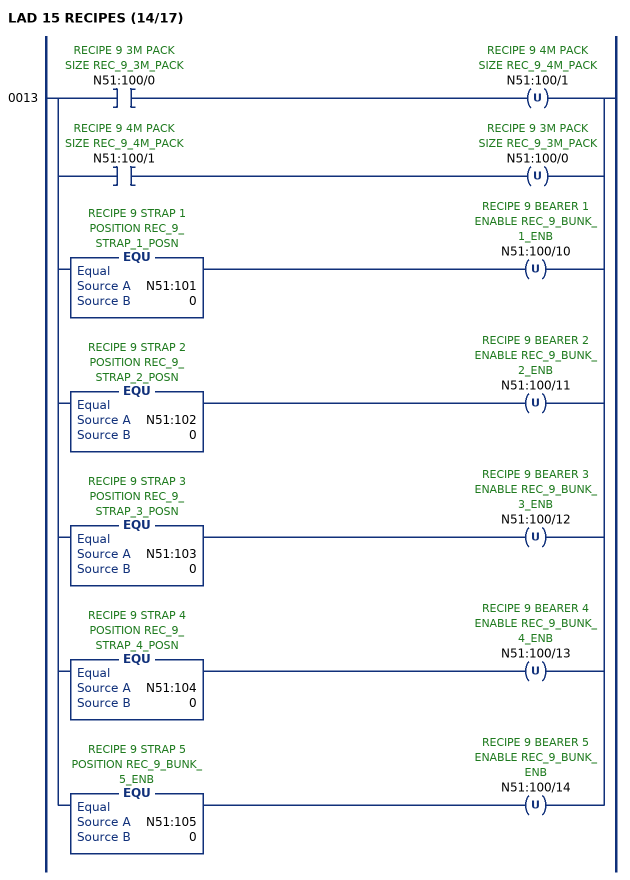
% Rung: 13 %
SOR BST XIC N51:100/0 OTU N51:100/1 NXB XIC N51:100/1 OTU N51:100/0 NXB EQU N51:101 0 OTU N51:100/10 NXB EQU N51:102 0 OTU N51:100/11 NXB EQU N51:103 0 OTU N51:100/12 NXB EQU N51:104 0 OTU N51:100/13 NXB EQU N51:105 0 OTU N51:100/14 BND EOR
%   N51:100/0  REC_9_3M_PACK  "RECIPE 9 3M PACK SIZE" %
%   N51:100/1  REC_9_4M_PACK  "RECIPE 9 4M PACK SIZE" %
%   N51:101  REC_9_STRAP_1_POSN  "RECIPE 9 STRAP 1 POSITION" %
%   N51:100/10  REC_9_BUNK_1_ENB  "RECIPE 9 BEARER 1 ENABLE" %
%   N51:102  REC_9_STRAP_2_POSN  "RECIPE 9 STRAP 2 POSITION" %
%   N51:100/11  REC_9_BUNK_2_ENB  "RECIPE 9 BEARER 2 ENABLE" %
%   N51:103  REC_9_STRAP_3_POSN  "RECIPE 9 STRAP 3 POSITION" %
%   N51:100/12  REC_9_BUNK_3_ENB  "RECIPE 9 BEARER 3 ENABLE" %
%   N51:104  REC_9_STRAP_4_POSN  "RECIPE 9 STRAP 4 POSITION" %
%   N51:100/13  REC_9_BUNK_4_ENB  "RECIPE 9 BEARER 4 ENABLE" %
%   N51:105  REC_9_BUNK_5_ENB  "RECIPE 9 STRAP 5 POSITION" %
%   N51:100/14  REC_9_BUNK_ENB  "RECIPE 9 BEARER 5 ENABLE" %

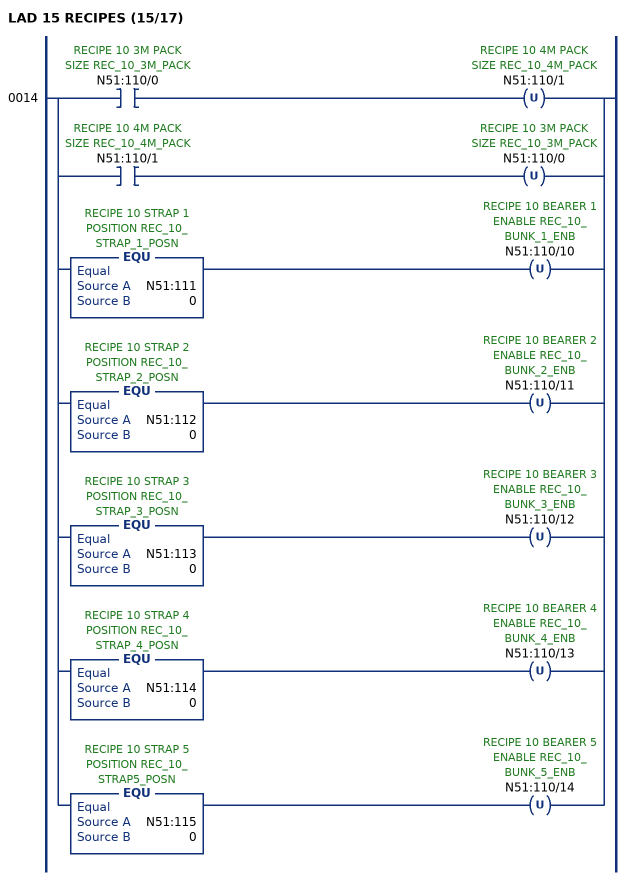
% Rung: 14 %
SOR BST XIC N51:110/0 OTU N51:110/1 NXB XIC N51:110/1 OTU N51:110/0 NXB EQU N51:111 0 OTU N51:110/10 NXB EQU N51:112 0 OTU N51:110/11 NXB EQU N51:113 0 OTU N51:110/12 NXB EQU N51:114 0 OTU N51:110/13 NXB EQU N51:115 0 OTU N51:110/14 BND EOR
%   N51:110/0  REC_10_3M_PACK  "RECIPE 10 3M PACK SIZE" %
%   N51:110/1  REC_10_4M_PACK  "RECIPE 10 4M PACK SIZE" %
%   N51:111  REC_10_STRAP_1_POSN  "RECIPE 10 STRAP 1 POSITION" %
%   N51:110/10  REC_10_BUNK_1_ENB  "RECIPE 10 BEARER 1 ENABLE" %
%   N51:112  REC_10_STRAP_2_POSN  "RECIPE 10 STRAP 2 POSITION" %
%   N51:110/11  REC_10_BUNK_2_ENB  "RECIPE 10 BEARER 2 ENABLE" %
%   N51:113  REC_10_STRAP_3_POSN  "RECIPE 10 STRAP 3 POSITION" %
%   N51:110/12  REC_10_BUNK_3_ENB  "RECIPE 10 BEARER 3 ENABLE" %
%   N51:114  REC_10_STRAP_4_POSN  "RECIPE 10 STRAP 4 POSITION" %
%   N51:110/13  REC_10_BUNK_4_ENB  "RECIPE 10 BEARER 4 ENABLE" %
%   N51:115  REC_10_STRAP5_POSN  "RECIPE 10 STRAP 5 POSITION" %
%   N51:110/14  REC_10_BUNK_5_ENB  "RECIPE 10 BEARER 5 ENABLE" %

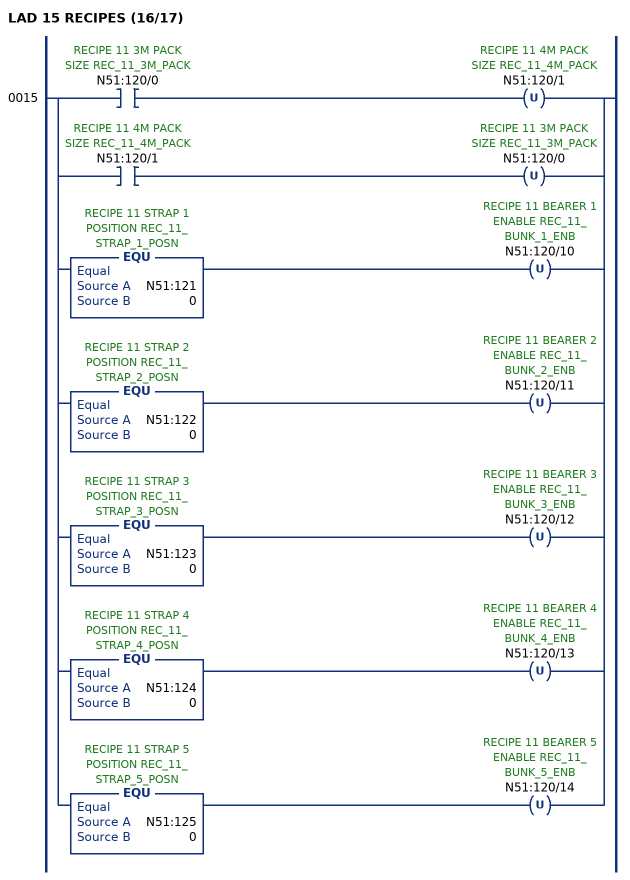
% Rung: 15 %
SOR BST XIC N51:120/0 OTU N51:120/1 NXB XIC N51:120/1 OTU N51:120/0 NXB EQU N51:121 0 OTU N51:120/10 NXB EQU N51:122 0 OTU N51:120/11 NXB EQU N51:123 0 OTU N51:120/12 NXB EQU N51:124 0 OTU N51:120/13 NXB EQU N51:125 0 OTU N51:120/14 BND EOR
%   N51:120/0  REC_11_3M_PACK  "RECIPE 11 3M PACK SIZE" %
%   N51:120/1  REC_11_4M_PACK  "RECIPE 11 4M PACK SIZE" %
%   N51:121  REC_11_STRAP_1_POSN  "RECIPE 11 STRAP 1 POSITION" %
%   N51:120/10  REC_11_BUNK_1_ENB  "RECIPE 11 BEARER 1 ENABLE" %
%   N51:122  REC_11_STRAP_2_POSN  "RECIPE 11 STRAP 2 POSITION" %
%   N51:120/11  REC_11_BUNK_2_ENB  "RECIPE 11 BEARER 2 ENABLE" %
%   N51:123  REC_11_STRAP_3_POSN  "RECIPE 11 STRAP 3 POSITION" %
%   N51:120/12  REC_11_BUNK_3_ENB  "RECIPE 11 BEARER 3 ENABLE" %
%   N51:124  REC_11_STRAP_4_POSN  "RECIPE 11 STRAP 4 POSITION" %
%   N51:120/13  REC_11_BUNK_4_ENB  "RECIPE 11 BEARER 4 ENABLE" %
%   N51:125  REC_11_STRAP_5_POSN  "RECIPE 11 STRAP 5 POSITION" %
%   N51:120/14  REC_11_BUNK_5_ENB  "RECIPE 11 BEARER 5 ENABLE" %

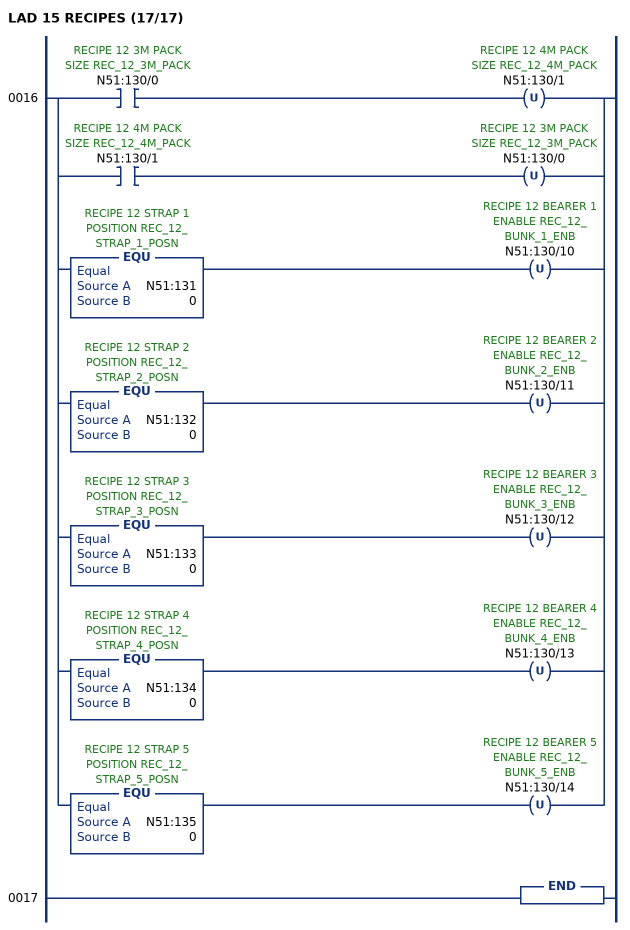
% Rung: 16 %
SOR BST XIC N51:130/0 OTU N51:130/1 NXB XIC N51:130/1 OTU N51:130/0 NXB EQU N51:131 0 OTU N51:130/10 NXB EQU N51:132 0 OTU N51:130/11 NXB EQU N51:133 0 OTU N51:130/12 NXB EQU N51:134 0 OTU N51:130/13 NXB EQU N51:135 0 OTU N51:130/14 BND EOR
%   N51:130/0  REC_12_3M_PACK  "RECIPE 12 3M PACK SIZE" %
%   N51:130/1  REC_12_4M_PACK  "RECIPE 12 4M PACK SIZE" %
%   N51:131  REC_12_STRAP_1_POSN  "RECIPE 12 STRAP 1 POSITION" %
%   N51:130/10  REC_12_BUNK_1_ENB  "RECIPE 12 BEARER 1 ENABLE" %
%   N51:132  REC_12_STRAP_2_POSN  "RECIPE 12 STRAP 2 POSITION" %
%   N51:130/11  REC_12_BUNK_2_ENB  "RECIPE 12 BEARER 2 ENABLE" %
%   N51:133  REC_12_STRAP_3_POSN  "RECIPE 12 STRAP 3 POSITION" %
%   N51:130/12  REC_12_BUNK_3_ENB  "RECIPE 12 BEARER 3 ENABLE" %
%   N51:134  REC_12_STRAP_4_POSN  "RECIPE 12 STRAP 4 POSITION" %
%   N51:130/13  REC_12_BUNK_4_ENB  "RECIPE 12 BEARER 4 ENABLE" %
%   N51:135  REC_12_STRAP_5_POSN  "RECIPE 12 STRAP 5 POSITION" %
%   N51:130/14  REC_12_BUNK_5_ENB  "RECIPE 12 BEARER 5 ENABLE" %
% Rung: 17 %
SOR END EOR

LADDER 16 "ENCODER"    % ENCODER %
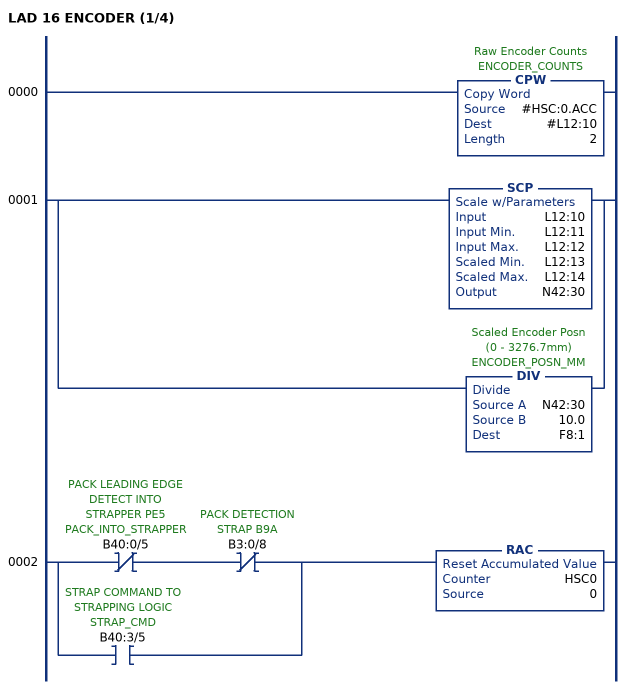
% Rung: 0 %
SOR CPW #HSC:0.ACC #L12:10 2 EOR
%   L12:10  ENCODER_COUNTS  "Raw Encoder Counts" %
% Rung: 1 %
SOR BST SCP L12:10 L12:11 L12:12 L12:13 L12:14 N42:30 NXB DIV N42:30 10.0 F8:1 BND EOR
%   L12:10  ENCODER_COUNTS  "Raw Encoder Counts" %
%   F8:1  ENCODER_POSN_MM  "Scaled Encoder Posn (0 - 3276.7mm)" %
% Rung: 2 %
SOR BST XIO B40:0/5 XIO B3:0/8 NXB XIC B40:3/5 BND RAC HSC0 0 EOR
%   B40:0/5  PACK_INTO_STRAPPER  "PACK LEADING EDGE DETECT INTO STRAPPER PE5" %
%   B3:0/8  B9A  "PACK DETECTION STRAP" %
%   B40:3/5  STRAP_CMD  "STRAP COMMAND TO STRAPPING LOGIC" %

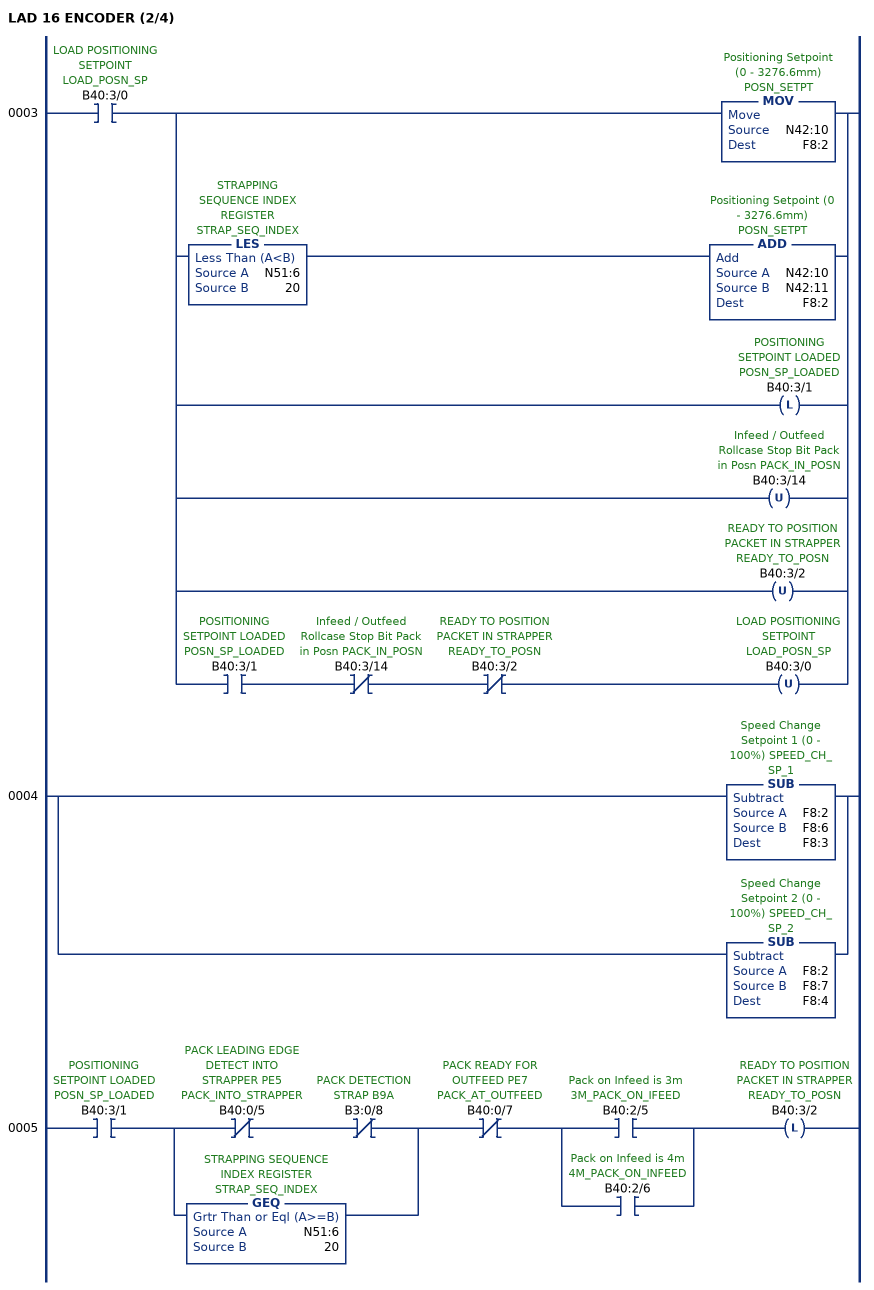
% Rung: 3 %
SOR XIC B40:3/0 BST MOV N42:10 F8:2 NXB LES N51:6 20 ADD N42:10 N42:11 F8:2 NXB OTL B40:3/1 NXB OTU B40:3/14 NXB OTU B40:3/2 NXB XIC B40:3/1 XIO B40:3/14 XIO B40:3/2 OTU B40:3/0 BND EOR
%   B40:3/0  LOAD_POSN_SP  "LOAD POSITIONING SETPOINT" %
%   N42:10  POSN_SETPOINT  "POSITIONING SETPOINT" %
%   F8:2  POSN_SETPT  "Positioning Setpoint (0 - 3276.6mm)" %
%   N51:6  STRAP_SEQ_INDEX  "STRAPPING SEQUENCE INDEX REGISTER" %
%   N42:11  POSN_SP_OFFSET  "Positioning Setpoint Offset" %
%   B40:3/1  POSN_SP_LOADED  "POSITIONING SETPOINT LOADED" %
%   B40:3/14  PACK_IN_POSN  "Infeed / Outfeed Rollcase Stop Bit Pack in Posn" %
%   B40:3/2  READY_TO_POSN  "READY TO POSITION PACKET IN STRAPPER" %
% Rung: 4 %
SOR BST SUB F8:2 F8:6 F8:3 NXB SUB F8:2 F8:7 F8:4 BND EOR
%   F8:2  POSN_SETPT  "Positioning Setpoint (0 - 3276.6mm)" %
%   F8:6  SP_CHANGE_FACT_1  "Speed Change Position Factor 1" %
%   F8:3  SPEED_CH_SP_1  "Speed Change Setpoint 1 (0 - 100%)" %
%   F8:7  SP_CHANGE_FACT_2  "Speed Change Positon Factor 2" %
%   F8:4  SPEED_CH_SP_2  "Speed Change Setpoint 2 (0 - 100%)" %
% Rung: 5 %
SOR XIC B40:3/1 BST XIO B40:0/5 XIO B3:0/8 NXB GEQ N51:6 20 BND XIO B40:0/7 BST XIC B40:2/5 NXB XIC B40:2/6 BND OTL B40:3/2 EOR
%   B40:3/1  POSN_SP_LOADED  "POSITIONING SETPOINT LOADED" %
%   B40:0/5  PACK_INTO_STRAPPER  "PACK LEADING EDGE DETECT INTO STRAPPER PE5" %
%   B3:0/8  B9A  "PACK DETECTION STRAP" %
%   N51:6  STRAP_SEQ_INDEX  "STRAPPING SEQUENCE INDEX REGISTER" %
%   B40:0/7  PACK_AT_OUTFEED  "PACK READY FOR OUTFEED PE7" %
%   B40:2/5  3M_PACK_ON_IFEED  "Pack on Infeed is 3m" %
%   B40:2/6  4M_PACK_ON_INFEED  "Pack on Infeed is 4m" %
%   B40:3/2  READY_TO_POSN  "READY TO POSITION PACKET IN STRAPPER" %

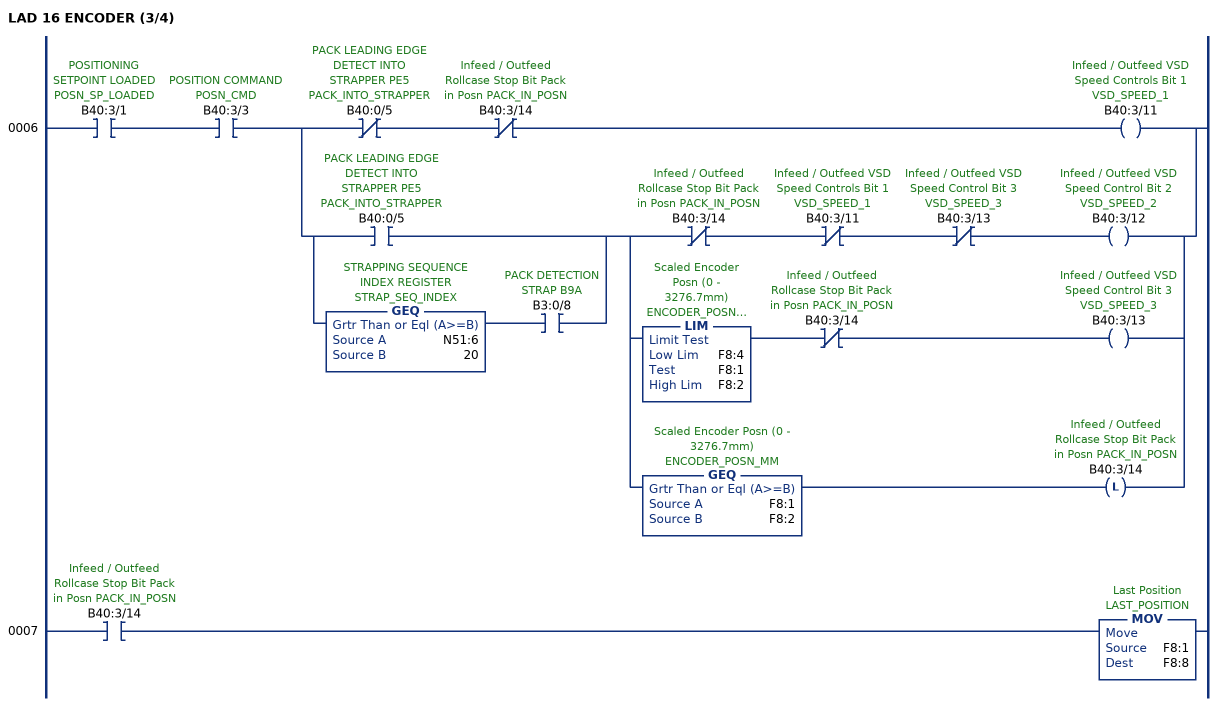
% Rung: 6 %
SOR XIC B40:3/1 XIC B40:3/3 BST XIO B40:0/5 XIO B40:3/14 OTE B40:3/11 NXB BST XIC B40:0/5 NXB GEQ N51:6 20 XIC B3:0/8 BND BST XIO B40:3/14 XIO B40:3/11 XIO B40:3/13 OTE B40:3/12 NXB LIM F8:4 F8:1 F8:2 XIO B40:3/14 OTE B40:3/13 NXB GEQ F8:1 F8:2 OTL B40:3/14 BND BND EOR
%   B40:3/1  POSN_SP_LOADED  "POSITIONING SETPOINT LOADED" %
%   B40:3/3  POSN_CMD  "POSITION COMMAND" %
%   B40:0/5  PACK_INTO_STRAPPER  "PACK LEADING EDGE DETECT INTO STRAPPER PE5" %
%   B40:3/14  PACK_IN_POSN  "Infeed / Outfeed Rollcase Stop Bit Pack in Posn" %
%   B40:3/11  VSD_SPEED_1  "Infeed / Outfeed VSD Speed Controls Bit 1" %
%   N51:6  STRAP_SEQ_INDEX  "STRAPPING SEQUENCE INDEX REGISTER" %
%   B3:0/8  B9A  "PACK DETECTION STRAP" %
%   B40:3/13  VSD_SPEED_3  "Infeed / Outfeed VSD Speed Control Bit 3" %
%   B40:3/12  VSD_SPEED_2  "Infeed / Outfeed VSD Speed Control Bit 2" %
%   F8:4  SPEED_CH_SP_2  "Speed Change Setpoint 2 (0 - 100%)" %
%   F8:1  ENCODER_POSN_MM  "Scaled Encoder Posn (0 - 3276.7mm)" %
%   F8:2  POSN_SETPT  "Positioning Setpoint (0 - 3276.6mm)" %
% Rung: 7 %
SOR XIC B40:3/14 MOV F8:1 F8:8 EOR
%   B40:3/14  PACK_IN_POSN  "Infeed / Outfeed Rollcase Stop Bit Pack in Posn" %
%   F8:1  ENCODER_POSN_MM  "Scaled Encoder Posn (0 - 3276.7mm)" %
%   F8:8  LAST_POSITION  "Last Position" %

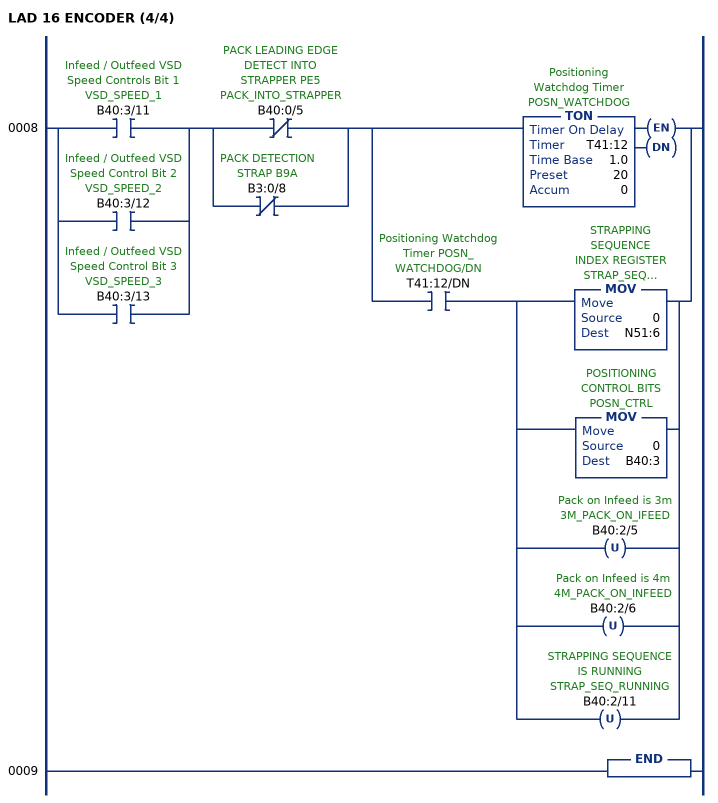
% Rung: 8 %
SOR BST XIC B40:3/11 NXB XIC B40:3/12 NXB XIC B40:3/13 BND BST XIO B40:0/5 NXB XIO B3:0/8 BND BST TON T41:12 1.0 20 0 NXB XIC T41:12/DN BST MOV 0 N51:6 NXB MOV 0 B40:3 NXB OTU B40:2/5 NXB OTU B40:2/6 NXB OTU B40:2/11 BND BND EOR
%   B40:3/11  VSD_SPEED_1  "Infeed / Outfeed VSD Speed Controls Bit 1" %
%   B40:3/12  VSD_SPEED_2  "Infeed / Outfeed VSD Speed Control Bit 2" %
%   B40:3/13  VSD_SPEED_3  "Infeed / Outfeed VSD Speed Control Bit 3" %
%   B40:0/5  PACK_INTO_STRAPPER  "PACK LEADING EDGE DETECT INTO STRAPPER PE5" %
%   B3:0/8  B9A  "PACK DETECTION STRAP" %
%   T41:12  POSN_WATCHDOG  "Positioning Watchdog Timer" %
%   N51:6  STRAP_SEQ_INDEX  "STRAPPING SEQUENCE INDEX REGISTER" %
%   B40:3  POSN_CTRL  "POSITIONING CONTROL BITS" %
%   B40:2/5  3M_PACK_ON_IFEED  "Pack on Infeed is 3m" %
%   B40:2/6  4M_PACK_ON_INFEED  "Pack on Infeed is 4m" %
%   B40:2/11  STRAP_SEQ_RUNNING  "STRAPPING SEQUENCE IS RUNNING" %
% Rung: 9 %
SOR END EOR

LADDER 17 "VSD"    % INFEED VSD'S %
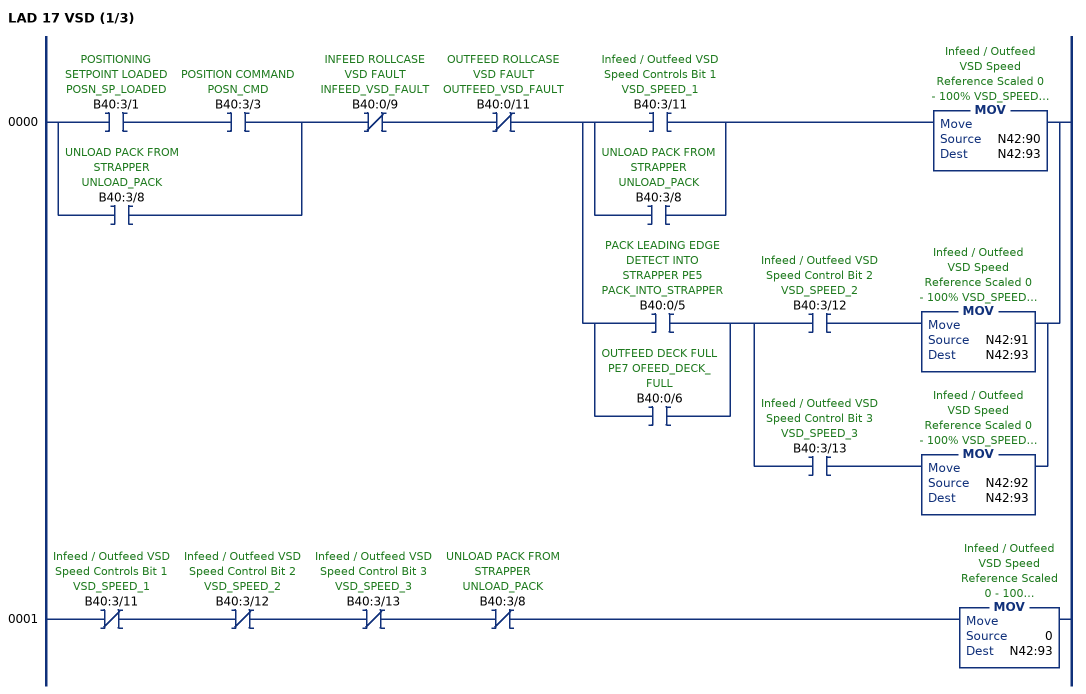
% Rung: 0 %
SOR BST XIC B40:3/1 XIC B40:3/3 NXB XIC B40:3/8 BND XIO B40:0/9 XIO B40:0/11 BST BST XIC B40:3/11 NXB XIC B40:3/8 BND MOV N42:90 N42:93 NXB BST XIC B40:0/5 NXB XIC B40:0/6 BND BST XIC B40:3/12 MOV N42:91 N42:93 NXB XIC B40:3/13 MOV N42:92 N42:93 BND BND EOR
%   B40:3/1  POSN_SP_LOADED  "POSITIONING SETPOINT LOADED" %
%   B40:3/3  POSN_CMD  "POSITION COMMAND" %
%   B40:3/8  UNLOAD_PACK  "UNLOAD PACK FROM STRAPPER" %
%   B40:0/9  INFEED_VSD_FAULT  "INFEED ROLLCASE VSD FAULT" %
%   B40:0/11  OUTFEED_VSD_FAULT  "OUTFEED ROLLCASE VSD FAULT" %
%   B40:3/11  VSD_SPEED_1  "Infeed / Outfeed VSD Speed Controls Bit 1" %
%   N42:90  VSD_SPEED_SP_1  "Infeed / Outfeed VSD Speed Setpoint 1 (0 - 100%)" %
%   N42:93  VSD_SPEED_REF  "Infeed / Outfeed VSD Speed Reference Scaled 0 - 100%" %
%   B40:0/5  PACK_INTO_STRAPPER  "PACK LEADING EDGE DETECT INTO STRAPPER PE5" %
%   B40:0/6  OFEED_DECK_FULL  "OUTFEED DECK FULL PE7" %
%   B40:3/12  VSD_SPEED_2  "Infeed / Outfeed VSD Speed Control Bit 2" %
%   N42:91  VSD_SPEED_SP_2  "Infeed / Outfeed VSD Speed Setpoint 2 (0 - 100%)" %
%   B40:3/13  VSD_SPEED_3  "Infeed / Outfeed VSD Speed Control Bit 3" %
%   N42:92  VSD_SPEED_SP_3  "Infeed / Outfeed VSD Speed Setpoint 3 (0 - 100%)" %
% Rung: 1 %
SOR XIO B40:3/11 XIO B40:3/12 XIO B40:3/13 XIO B40:3/8 MOV 0 N42:93 EOR
%   B40:3/11  VSD_SPEED_1  "Infeed / Outfeed VSD Speed Controls Bit 1" %
%   B40:3/12  VSD_SPEED_2  "Infeed / Outfeed VSD Speed Control Bit 2" %
%   B40:3/13  VSD_SPEED_3  "Infeed / Outfeed VSD Speed Control Bit 3" %
%   B40:3/8  UNLOAD_PACK  "UNLOAD PACK FROM STRAPPER" %
%   N42:93  VSD_SPEED_REF  "Infeed / Outfeed VSD Speed Reference Scaled 0 - 100%" %

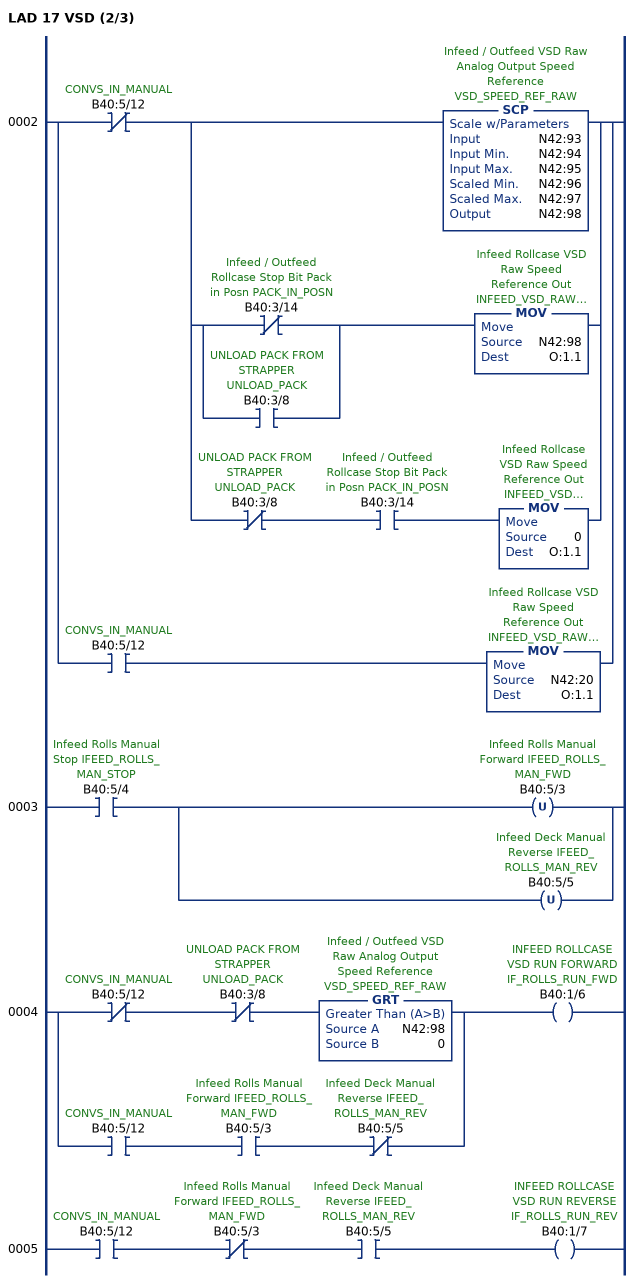
% Rung: 2 %
SOR BST XIO B40:5/12 BST BST SCP N42:93 N42:94 N42:95 N42:96 N42:97 N42:98 NXB BST XIO B40:3/14 NXB XIC B40:3/8 BND MOV N42:98 O:1.1 BND NXB XIO B40:3/8 XIC B40:3/14 MOV 0 O:1.1 BND NXB XIC B40:5/12 MOV N42:20 O:1.1 BND EOR
%   B40:5/12  CONVS_IN_MANUAL %
%   N42:93  VSD_SPEED_REF  "Infeed / Outfeed VSD Speed Reference Scaled 0 - 100%" %
%   N42:94  "Infeed / Outfeed VSD Scaled Input Max" %
%   N42:95  "Infeed / Outfeed VSD Scaled Input Min" %
%   N42:96  "Infeed / Outfeed VSD Scaled Output Min To Analog" %
%   N42:97  "Infeed / Outfeed VSD Scaled Output Max To Analog" %
%   N42:98  VSD_SPEED_REF_RAW  "Infeed / Outfeed VSD Raw Analog Output Speed Reference" %
%   B40:3/14  PACK_IN_POSN  "Infeed / Outfeed Rollcase Stop Bit Pack in Posn" %
%   B40:3/8  UNLOAD_PACK  "UNLOAD PACK FROM STRAPPER" %
%   O:1.1  INFEED_VSD_RAW_OUT  "Infeed Rollcase VSD Raw Speed Reference Out" %
%   N42:20  VSD_MAN_SPEED_SP  "VSD MANUAL SPEED SETPOINT" %
% Rung: 3 %
SOR XIC B40:5/4 BST OTU B40:5/3 NXB OTU B40:5/5 BND EOR
%   B40:5/4  IFEED_ROLLS_MAN_STOP  "Infeed Rolls Manual Stop" %
%   B40:5/3  IFEED_ROLLS_MAN_FWD  "Infeed Rolls Manual Forward" %
%   B40:5/5  IFEED_ROLLS_MAN_REV  "Infeed Deck Manual Reverse" %
% Rung: 4 %
SOR BST XIO B40:5/12 XIO B40:3/8 GRT N42:98 0 NXB XIC B40:5/12 XIC B40:5/3 XIO B40:5/5 BND OTE B40:1/6 EOR
%   B40:5/12  CONVS_IN_MANUAL %
%   B40:3/8  UNLOAD_PACK  "UNLOAD PACK FROM STRAPPER" %
%   N42:98  VSD_SPEED_REF_RAW  "Infeed / Outfeed VSD Raw Analog Output Speed Reference" %
%   B40:5/3  IFEED_ROLLS_MAN_FWD  "Infeed Rolls Manual Forward" %
%   B40:5/5  IFEED_ROLLS_MAN_REV  "Infeed Deck Manual Reverse" %
%   B40:1/6  IF_ROLLS_RUN_FWD  "INFEED ROLLCASE VSD RUN FORWARD" %
% Rung: 5 %
SOR XIC B40:5/12 XIO B40:5/3 XIC B40:5/5 OTE B40:1/7 EOR
%   B40:5/12  CONVS_IN_MANUAL %
%   B40:5/3  IFEED_ROLLS_MAN_FWD  "Infeed Rolls Manual Forward" %
%   B40:5/5  IFEED_ROLLS_MAN_REV  "Infeed Deck Manual Reverse" %
%   B40:1/7  IF_ROLLS_RUN_REV  "INFEED ROLLCASE VSD RUN REVERSE" %

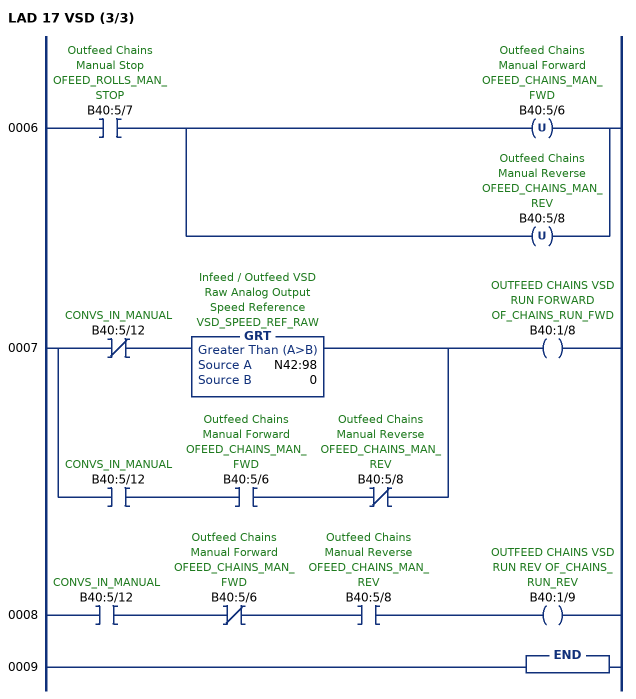
% Rung: 6 %
SOR XIC B40:5/7 BST OTU B40:5/6 NXB OTU B40:5/8 BND EOR
%   B40:5/7  OFEED_ROLLS_MAN_STOP  "Outfeed Chains Manual Stop" %
%   B40:5/6  OFEED_CHAINS_MAN_FWD  "Outfeed Chains Manual Forward" %
%   B40:5/8  OFEED_CHAINS_MAN_REV  "Outfeed Chains Manual Reverse" %
% Rung: 7 %
SOR BST XIO B40:5/12 GRT N42:98 0 NXB XIC B40:5/12 XIC B40:5/6 XIO B40:5/8 BND OTE B40:1/8 EOR
%   B40:5/12  CONVS_IN_MANUAL %
%   N42:98  VSD_SPEED_REF_RAW  "Infeed / Outfeed VSD Raw Analog Output Speed Reference" %
%   B40:5/6  OFEED_CHAINS_MAN_FWD  "Outfeed Chains Manual Forward" %
%   B40:5/8  OFEED_CHAINS_MAN_REV  "Outfeed Chains Manual Reverse" %
%   B40:1/8  OF_CHAINS_RUN_FWD  "OUTFEED CHAINS VSD RUN FORWARD" %
% Rung: 8 %
SOR XIC B40:5/12 XIO B40:5/6 XIC B40:5/8 OTE B40:1/9 EOR
%   B40:5/12  CONVS_IN_MANUAL %
%   B40:5/6  OFEED_CHAINS_MAN_FWD  "Outfeed Chains Manual Forward" %
%   B40:5/8  OFEED_CHAINS_MAN_REV  "Outfeed Chains Manual Reverse" %
%   B40:1/9  OF_CHAINS_RUN_REV  "OUTFEED CHAINS VSD RUN REV" %
% Rung: 9 %
SOR END EOR

LADDER 18 "RECIPE SEQ"
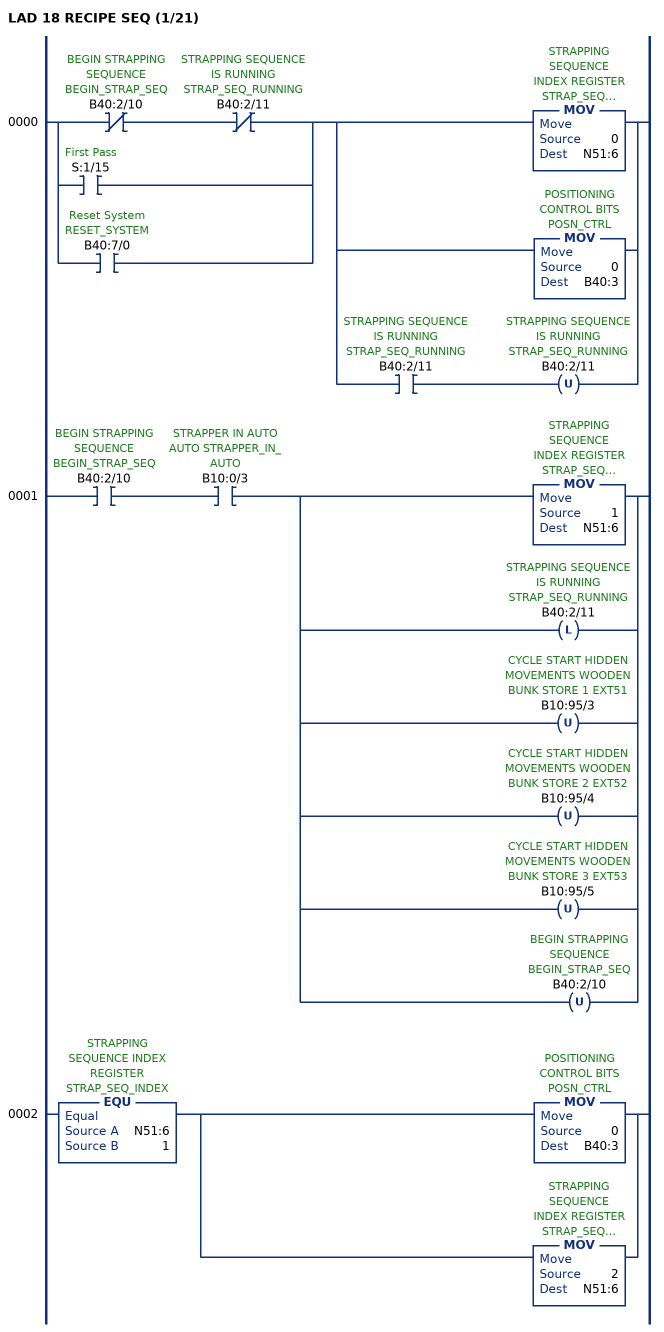
% Rung: 0 %
SOR BST XIO B40:2/10 XIO B40:2/11 NXB XIC S:1/15 NXB XIC B40:7/0 BND BST MOV 0 N51:6 NXB MOV 0 B40:3 NXB XIC B40:2/11 OTU B40:2/11 BND EOR
%   B40:2/10  BEGIN_STRAP_SEQ  "BEGIN STRAPPING SEQUENCE" %
%   B40:2/11  STRAP_SEQ_RUNNING  "STRAPPING SEQUENCE IS RUNNING" %
%   S:1/15  "First Pass" %
%   B40:7/0  RESET_SYSTEM  "Reset System" %
%   N51:6  STRAP_SEQ_INDEX  "STRAPPING SEQUENCE INDEX REGISTER" %
%   B40:3  POSN_CTRL  "POSITIONING CONTROL BITS" %
% Rung: 1 %
SOR XIC B40:2/10 XIC B10:0/3 BST MOV 1 N51:6 NXB OTL B40:2/11 NXB OTU B10:95/3 NXB OTU B10:95/4 NXB OTU B10:95/5 NXB OTU B40:2/10 BND EOR
%   B40:2/10  BEGIN_STRAP_SEQ  "BEGIN STRAPPING SEQUENCE" %
%   B10:0/3  STRAPPER_IN_AUTO  "STRAPPER IN AUTO AUTO" %
%   N51:6  STRAP_SEQ_INDEX  "STRAPPING SEQUENCE INDEX REGISTER" %
%   B40:2/11  STRAP_SEQ_RUNNING  "STRAPPING SEQUENCE IS RUNNING" %
%   B10:95/3  EXT51  "CYCLE START HIDDEN MOVEMENTS WOODEN BUNK STORE 1" %
%   B10:95/4  EXT52  "CYCLE START HIDDEN MOVEMENTS WOODEN BUNK STORE 2" %
%   B10:95/5  EXT53  "CYCLE START HIDDEN MOVEMENTS WOODEN BUNK STORE 3" %
% Rung: 2 %
SOR EQU N51:6 1 BST MOV 0 B40:3 NXB MOV 2 N51:6 BND EOR
%   N51:6  STRAP_SEQ_INDEX  "STRAPPING SEQUENCE INDEX REGISTER" %
%   B40:3  POSN_CTRL  "POSITIONING CONTROL BITS" %

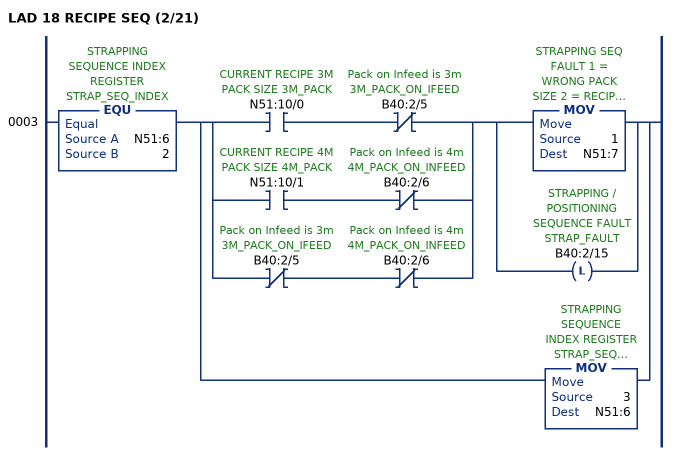
% Rung: 3 %
SOR EQU N51:6 2 BST BST XIC N51:10/0 XIO B40:2/5 NXB XIC N51:10/1 XIO B40:2/6 NXB XIO B40:2/5 XIO B40:2/6 BND BST MOV 1 N51:7 NXB OTL B40:2/15 BND NXB MOV 3 N51:6 BND EOR
%   N51:6  STRAP_SEQ_INDEX  "STRAPPING SEQUENCE INDEX REGISTER" %
%   N51:10/0  3M_PACK  "CURRENT RECIPE 3M PACK SIZE" %
%   B40:2/5  3M_PACK_ON_IFEED  "Pack on Infeed is 3m" %
%   N51:10/1  4M_PACK  "CURRENT RECIPE 4M PACK SIZE" %
%   B40:2/6  4M_PACK_ON_INFEED  "Pack on Infeed is 4m" %
%   N51:7  STRAP_SEQ_FLT  "STRAPPING SEQ FAULT 1 = WRONG PACK SIZE 2 = RECIPE FAULT 3 = POSNING FAULT 4 = STRAPPING FAULT" %
%   B40:2/15  STRAP_FAULT  "STRAPPING / POSITIONING SEQUENCE FAULT" %

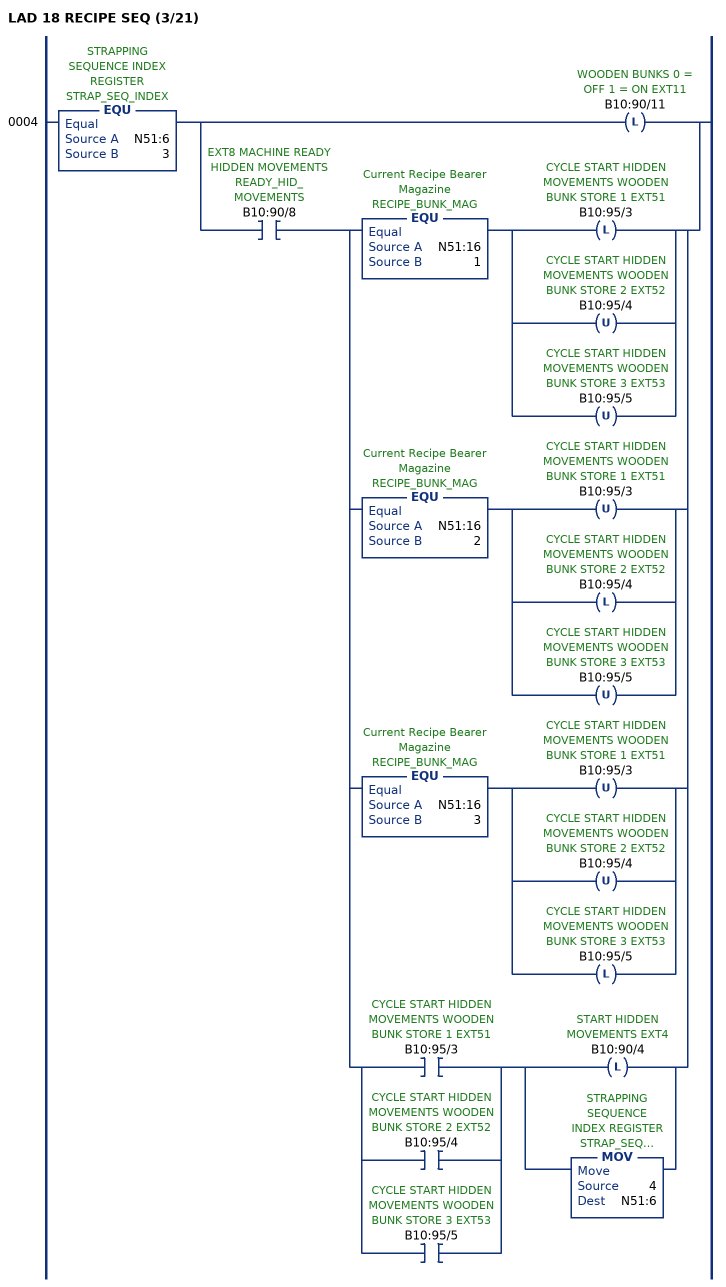
% Rung: 4 %
SOR EQU N51:6 3 BST OTL B10:90/11 NXB XIC B10:90/8 BST EQU N51:16 1 BST OTL B10:95/3 NXB OTU B10:95/4 NXB OTU B10:95/5 BND NXB EQU N51:16 2 BST OTU B10:95/3 NXB OTL B10:95/4 NXB OTU B10:95/5 BND NXB EQU N51:16 3 BST OTU B10:95/3 NXB OTU B10:95/4 NXB OTL B10:95/5 BND NXB BST XIC B10:95/3 NXB XIC B10:95/4 NXB XIC B10:95/5 BND BST OTL B10:90/4 NXB MOV 4 N51:6 BND BND BND EOR
%   N51:6  STRAP_SEQ_INDEX  "STRAPPING SEQUENCE INDEX REGISTER" %
%   B10:90/11  EXT11  "WOODEN BUNKS 0 = OFF 1 = ON" %
%   B10:90/8  READY_HID_MOVEMENTS  "EXT8 MACHINE READY HIDDEN MOVEMENTS" %
%   N51:16  RECIPE_BUNK_MAG  "Current Recipe Bearer Magazine" %
%   B10:95/3  EXT51  "CYCLE START HIDDEN MOVEMENTS WOODEN BUNK STORE 1" %
%   B10:95/4  EXT52  "CYCLE START HIDDEN MOVEMENTS WOODEN BUNK STORE 2" %
%   B10:95/5  EXT53  "CYCLE START HIDDEN MOVEMENTS WOODEN BUNK STORE 3" %
%   B10:90/4  EXT4  "START HIDDEN MOVEMENTS" %

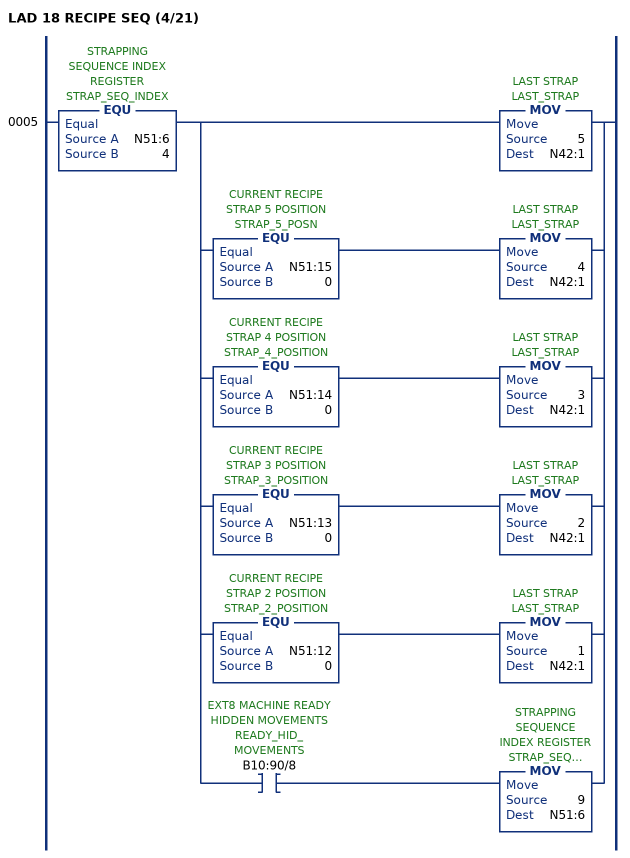
% Rung: 5 %
SOR EQU N51:6 4 BST MOV 5 N42:1 NXB EQU N51:15 0 MOV 4 N42:1 NXB EQU N51:14 0 MOV 3 N42:1 NXB EQU N51:13 0 MOV 2 N42:1 NXB EQU N51:12 0 MOV 1 N42:1 NXB XIC B10:90/8 MOV 9 N51:6 BND EOR
%   N51:6  STRAP_SEQ_INDEX  "STRAPPING SEQUENCE INDEX REGISTER" %
%   N42:1  LAST_STRAP  "LAST STRAP" %
%   N51:15  STRAP_5_POSN  "CURRENT RECIPE STRAP 5 POSITION" %
%   N51:14  STRAP_4_POSITION  "CURRENT RECIPE STRAP 4 POSITION" %
%   N51:13  STRAP_3_POSITION  "CURRENT RECIPE STRAP 3 POSITION" %
%   N51:12  STRAP_2_POSITION  "CURRENT RECIPE STRAP 2 POSITION" %
%   B10:90/8  READY_HID_MOVEMENTS  "EXT8 MACHINE READY HIDDEN MOVEMENTS" %

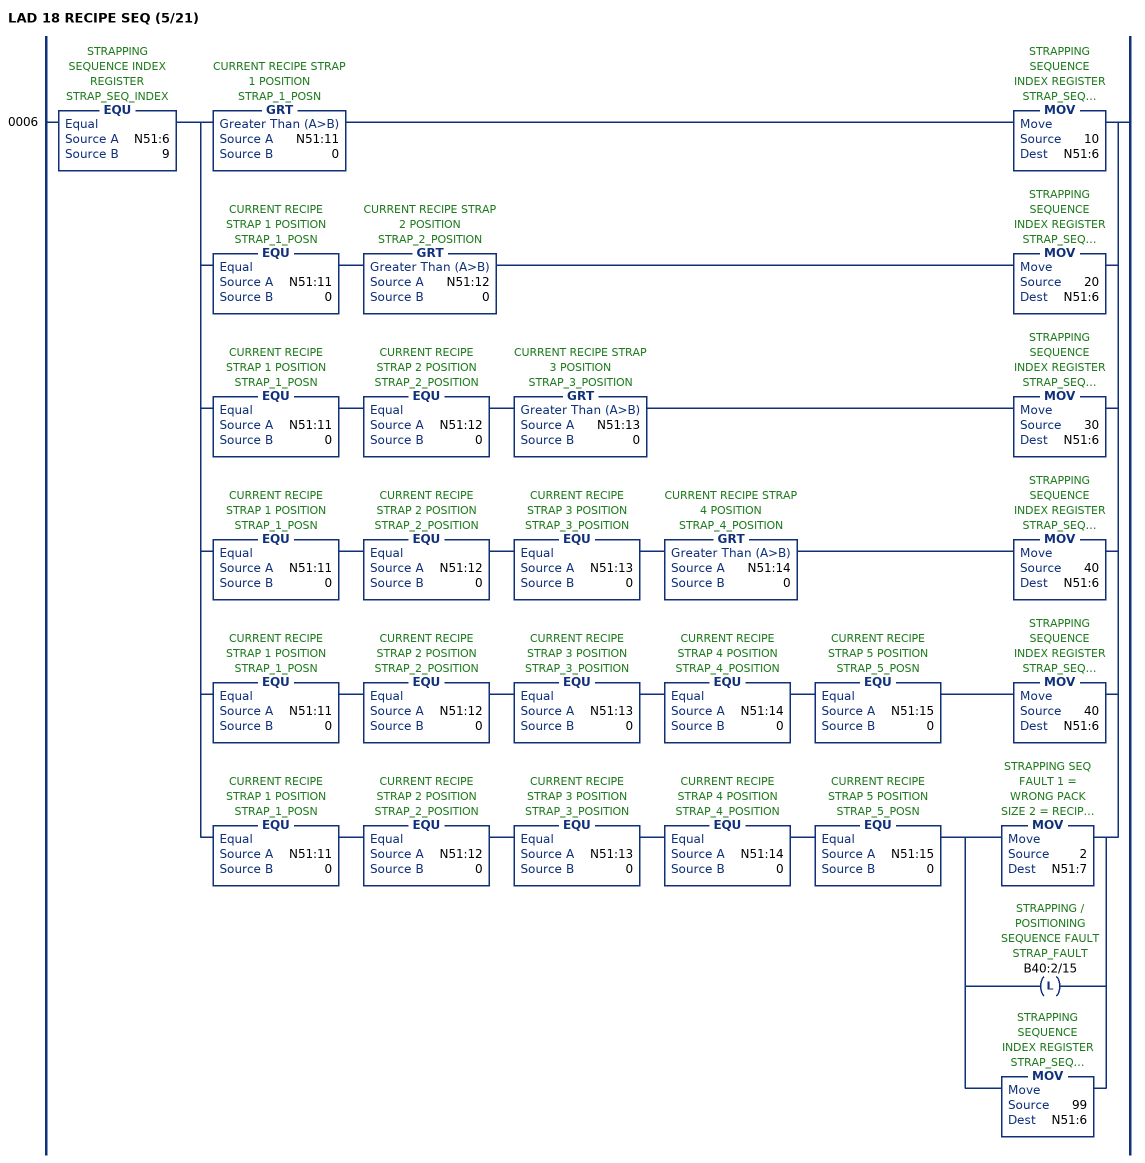
% Rung: 6 %
SOR EQU N51:6 9 BST GRT N51:11 0 MOV 10 N51:6 NXB EQU N51:11 0 GRT N51:12 0 MOV 20 N51:6 NXB EQU N51:11 0 EQU N51:12 0 GRT N51:13 0 MOV 30 N51:6 NXB EQU N51:11 0 EQU N51:12 0 EQU N51:13 0 GRT N51:14 0 MOV 40 N51:6 NXB EQU N51:11 0 EQU N51:12 0 EQU N51:13 0 EQU N51:14 0 EQU N51:15 0 MOV 40 N51:6 NXB EQU N51:11 0 EQU N51:12 0 EQU N51:13 0 EQU N51:14 0 EQU N51:15 0 BST MOV 2 N51:7 NXB OTL B40:2/15 NXB MOV 99 N51:6 BND BND EOR
%   N51:6  STRAP_SEQ_INDEX  "STRAPPING SEQUENCE INDEX REGISTER" %
%   N51:11  STRAP_1_POSN  "CURRENT RECIPE STRAP 1 POSITION" %
%   N51:12  STRAP_2_POSITION  "CURRENT RECIPE STRAP 2 POSITION" %
%   N51:13  STRAP_3_POSITION  "CURRENT RECIPE STRAP 3 POSITION" %
%   N51:14  STRAP_4_POSITION  "CURRENT RECIPE STRAP 4 POSITION" %
%   N51:15  STRAP_5_POSN  "CURRENT RECIPE STRAP 5 POSITION" %
%   N51:7  STRAP_SEQ_FLT  "STRAPPING SEQ FAULT 1 = WRONG PACK SIZE 2 = RECIPE FAULT 3 = POSNING FAULT 4 = STRAPPING FAULT" %
%   B40:2/15  STRAP_FAULT  "STRAPPING / POSITIONING SEQUENCE FAULT" %

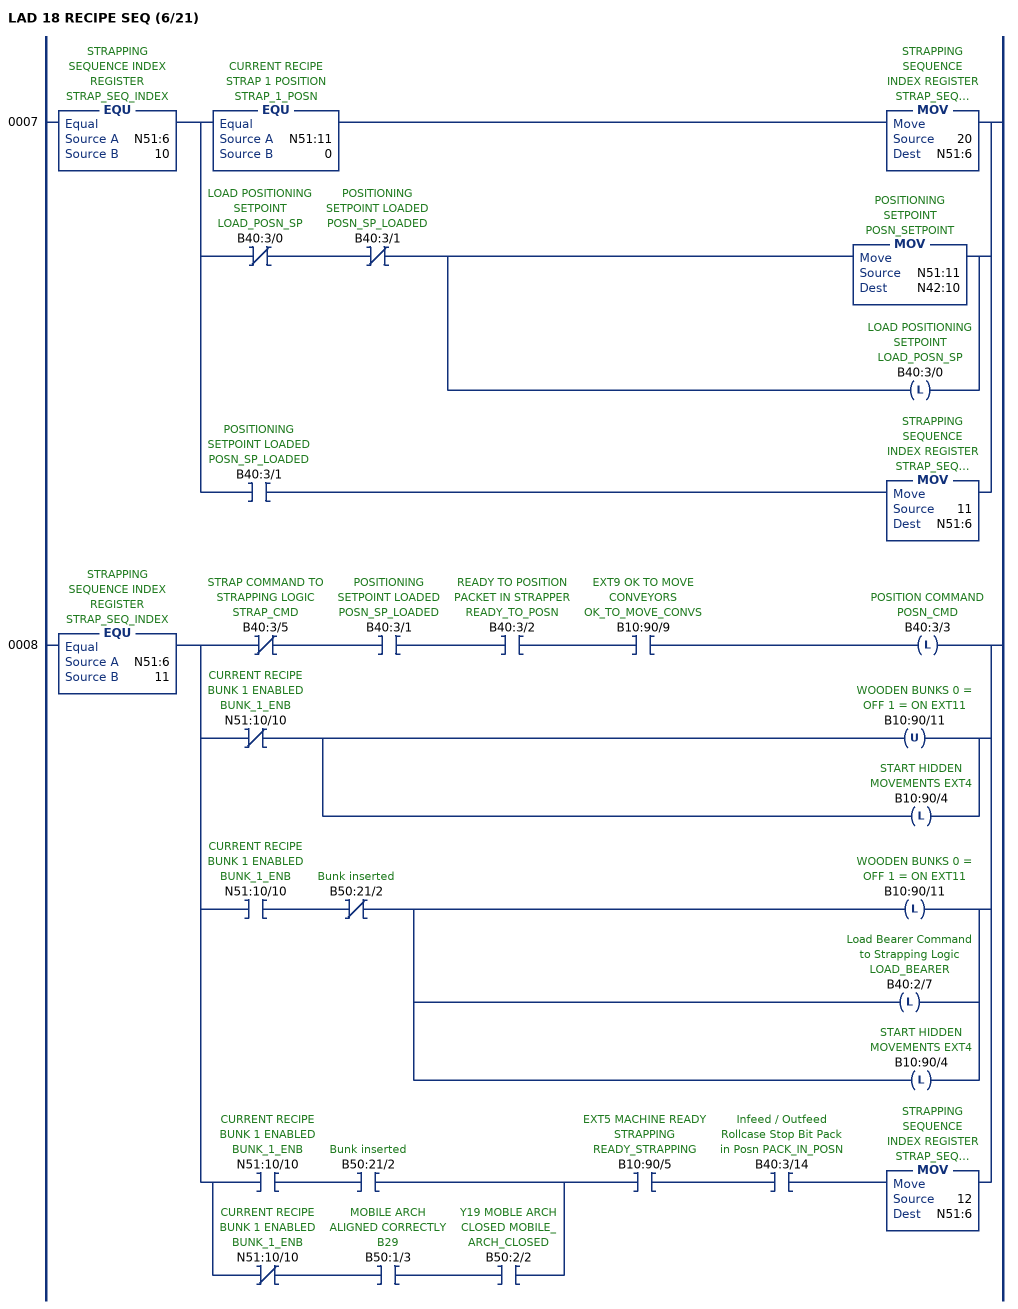
% Rung: 7 %
SOR EQU N51:6 10 BST EQU N51:11 0 MOV 20 N51:6 NXB XIO B40:3/0 XIO B40:3/1 BST MOV N51:11 N42:10 NXB OTL B40:3/0 BND NXB XIC B40:3/1 MOV 11 N51:6 BND EOR
%   N51:6  STRAP_SEQ_INDEX  "STRAPPING SEQUENCE INDEX REGISTER" %
%   N51:11  STRAP_1_POSN  "CURRENT RECIPE STRAP 1 POSITION" %
%   B40:3/0  LOAD_POSN_SP  "LOAD POSITIONING SETPOINT" %
%   B40:3/1  POSN_SP_LOADED  "POSITIONING SETPOINT LOADED" %
%   N42:10  POSN_SETPOINT  "POSITIONING SETPOINT" %
% Rung: 8 %
SOR EQU N51:6 11 BST XIO B40:3/5 XIC B40:3/1 XIC B40:3/2 XIC B10:90/9 OTL B40:3/3 NXB XIO N51:10/10 BST OTU B10:90/11 NXB OTL B10:90/4 BND NXB XIC N51:10/10 XIO B50:21/2 BST OTL B10:90/11 NXB OTL B40:2/7 NXB OTL B10:90/4 BND NXB BST XIC N51:10/10 XIC B50:21/2 NXB XIO N51:10/10 XIC B50:1/3 XIC B50:2/2 BND XIC B10:90/5 XIC B40:3/14 MOV 12 N51:6 BND EOR
%   N51:6  STRAP_SEQ_INDEX  "STRAPPING SEQUENCE INDEX REGISTER" %
%   B40:3/5  STRAP_CMD  "STRAP COMMAND TO STRAPPING LOGIC" %
%   B40:3/1  POSN_SP_LOADED  "POSITIONING SETPOINT LOADED" %
%   B40:3/2  READY_TO_POSN  "READY TO POSITION PACKET IN STRAPPER" %
%   B10:90/9  OK_TO_MOVE_CONVS  "EXT9 OK TO MOVE CONVEYORS" %
%   B40:3/3  POSN_CMD  "POSITION COMMAND" %
%   N51:10/10  BUNK_1_ENB  "CURRENT RECIPE BUNK 1 ENABLED" %
%   B10:90/11  EXT11  "WOODEN BUNKS 0 = OFF 1 = ON" %
%   B10:90/4  EXT4  "START HIDDEN MOVEMENTS" %
%   B50:21/2  "Bunk inserted" %
%   B40:2/7  LOAD_BEARER  "Load Bearer Command to Strapping Logic" %
%   B50:1/3  B29  "MOBILE ARCH ALIGNED CORRECTLY" %
%   B50:2/2  MOBILE_ARCH_CLOSED  "Y19 MOBLE ARCH CLOSED" %
%   B10:90/5  READY_STRAPPING  "EXT5 MACHINE READY STRAPPING" %
%   B40:3/14  PACK_IN_POSN  "Infeed / Outfeed Rollcase Stop Bit Pack in Posn" %

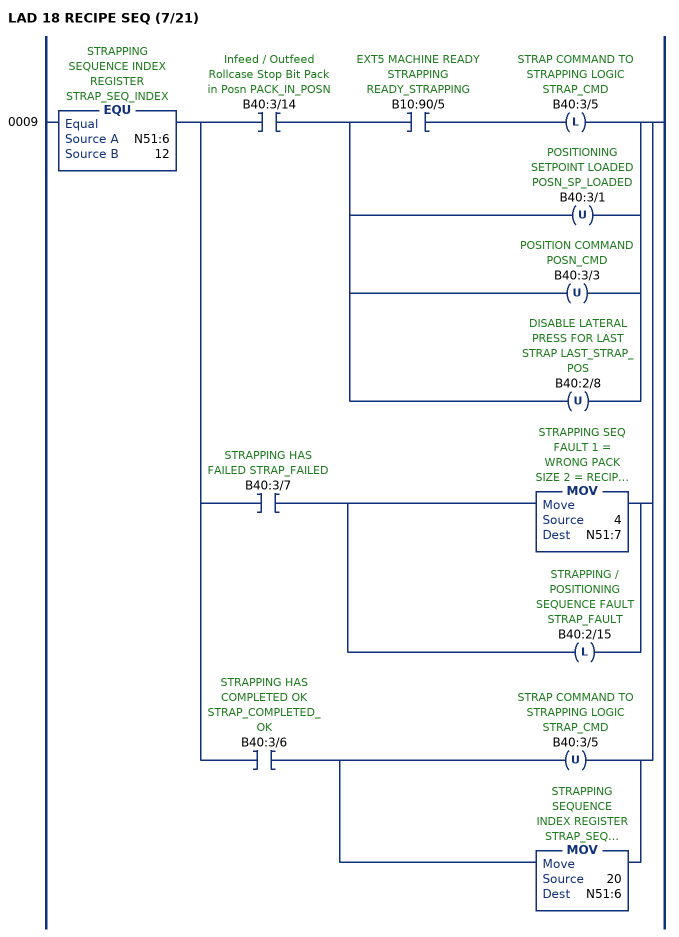
% Rung: 9 %
SOR EQU N51:6 12 BST XIC B40:3/14 BST XIC B10:90/5 OTL B40:3/5 NXB OTU B40:3/1 NXB OTU B40:3/3 NXB OTU B40:2/8 BND NXB XIC B40:3/7 BST MOV 4 N51:7 NXB OTL B40:2/15 BND NXB XIC B40:3/6 BST OTU B40:3/5 NXB MOV 20 N51:6 BND BND EOR
%   N51:6  STRAP_SEQ_INDEX  "STRAPPING SEQUENCE INDEX REGISTER" %
%   B40:3/14  PACK_IN_POSN  "Infeed / Outfeed Rollcase Stop Bit Pack in Posn" %
%   B10:90/5  READY_STRAPPING  "EXT5 MACHINE READY STRAPPING" %
%   B40:3/5  STRAP_CMD  "STRAP COMMAND TO STRAPPING LOGIC" %
%   B40:3/1  POSN_SP_LOADED  "POSITIONING SETPOINT LOADED" %
%   B40:3/3  POSN_CMD  "POSITION COMMAND" %
%   B40:2/8  LAST_STRAP_POS  "DISABLE LATERAL PRESS FOR LAST STRAP" %
%   B40:3/7  STRAP_FAILED  "STRAPPING HAS FAILED" %
%   N51:7  STRAP_SEQ_FLT  "STRAPPING SEQ FAULT 1 = WRONG PACK SIZE 2 = RECIPE FAULT 3 = POSNING FAULT 4 = STRAPPING FAULT" %
%   B40:2/15  STRAP_FAULT  "STRAPPING / POSITIONING SEQUENCE FAULT" %
%   B40:3/6  STRAP_COMPLETED_OK  "STRAPPING HAS COMPLETED OK" %

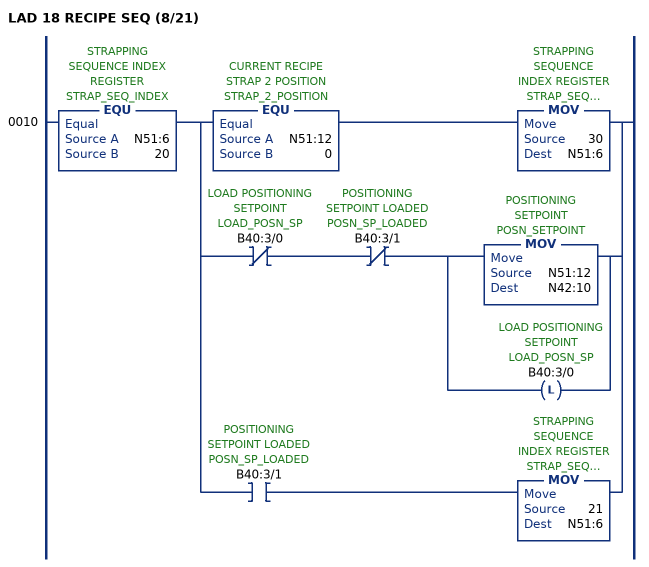
% Rung: 10 %
SOR EQU N51:6 20 BST EQU N51:12 0 MOV 30 N51:6 NXB XIO B40:3/0 XIO B40:3/1 BST MOV N51:12 N42:10 NXB OTL B40:3/0 BND NXB XIC B40:3/1 MOV 21 N51:6 BND EOR
%   N51:6  STRAP_SEQ_INDEX  "STRAPPING SEQUENCE INDEX REGISTER" %
%   N51:12  STRAP_2_POSITION  "CURRENT RECIPE STRAP 2 POSITION" %
%   B40:3/0  LOAD_POSN_SP  "LOAD POSITIONING SETPOINT" %
%   B40:3/1  POSN_SP_LOADED  "POSITIONING SETPOINT LOADED" %
%   N42:10  POSN_SETPOINT  "POSITIONING SETPOINT" %

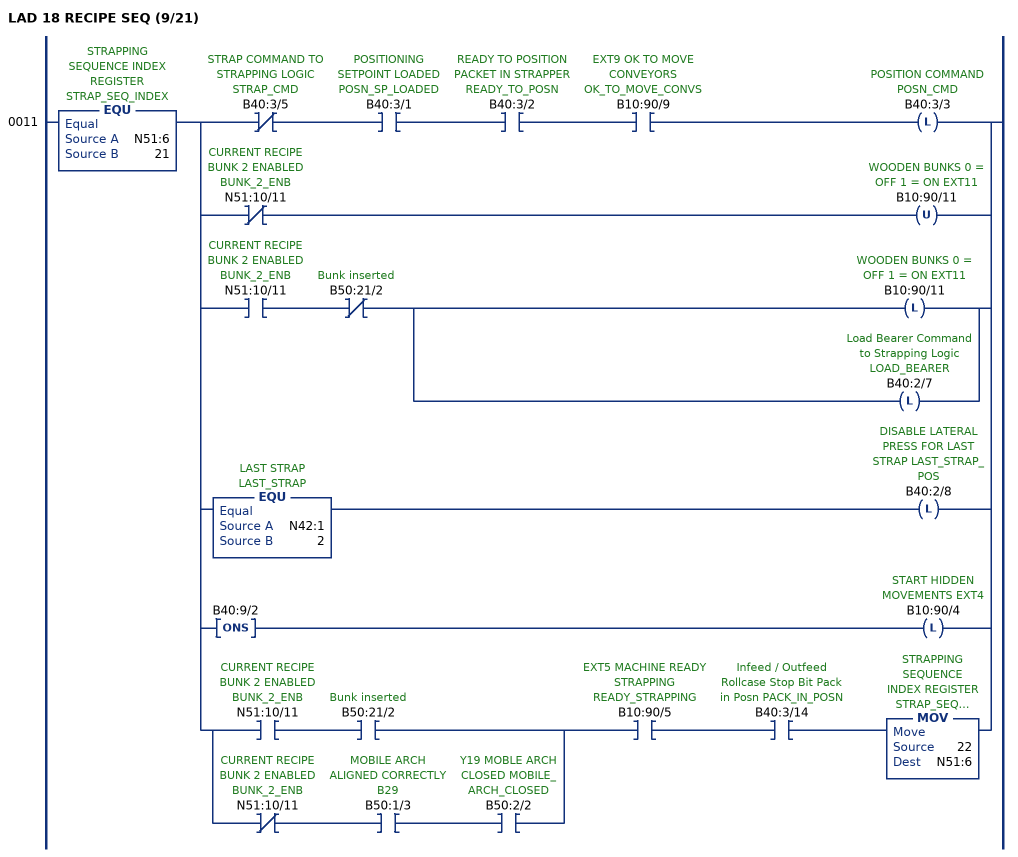
% Rung: 11 %
SOR EQU N51:6 21 BST XIO B40:3/5 XIC B40:3/1 XIC B40:3/2 XIC B10:90/9 OTL B40:3/3 NXB XIO N51:10/11 OTU B10:90/11 NXB XIC N51:10/11 XIO B50:21/2 BST OTL B10:90/11 NXB OTL B40:2/7 BND NXB EQU N42:1 2 OTL B40:2/8 NXB ONS B40:9/2 OTL B10:90/4 NXB BST XIC N51:10/11 XIC B50:21/2 NXB XIO N51:10/11 XIC B50:1/3 XIC B50:2/2 BND XIC B10:90/5 XIC B40:3/14 MOV 22 N51:6 BND EOR
%   N51:6  STRAP_SEQ_INDEX  "STRAPPING SEQUENCE INDEX REGISTER" %
%   B40:3/5  STRAP_CMD  "STRAP COMMAND TO STRAPPING LOGIC" %
%   B40:3/1  POSN_SP_LOADED  "POSITIONING SETPOINT LOADED" %
%   B40:3/2  READY_TO_POSN  "READY TO POSITION PACKET IN STRAPPER" %
%   B10:90/9  OK_TO_MOVE_CONVS  "EXT9 OK TO MOVE CONVEYORS" %
%   B40:3/3  POSN_CMD  "POSITION COMMAND" %
%   N51:10/11  BUNK_2_ENB  "CURRENT RECIPE BUNK 2 ENABLED" %
%   B10:90/11  EXT11  "WOODEN BUNKS 0 = OFF 1 = ON" %
%   B50:21/2  "Bunk inserted" %
%   B40:2/7  LOAD_BEARER  "Load Bearer Command to Strapping Logic" %
%   N42:1  LAST_STRAP  "LAST STRAP" %
%   B40:2/8  LAST_STRAP_POS  "DISABLE LATERAL PRESS FOR LAST STRAP" %
%   B10:90/4  EXT4  "START HIDDEN MOVEMENTS" %
%   B50:1/3  B29  "MOBILE ARCH ALIGNED CORRECTLY" %
%   B50:2/2  MOBILE_ARCH_CLOSED  "Y19 MOBLE ARCH CLOSED" %
%   B10:90/5  READY_STRAPPING  "EXT5 MACHINE READY STRAPPING" %
%   B40:3/14  PACK_IN_POSN  "Infeed / Outfeed Rollcase Stop Bit Pack in Posn" %

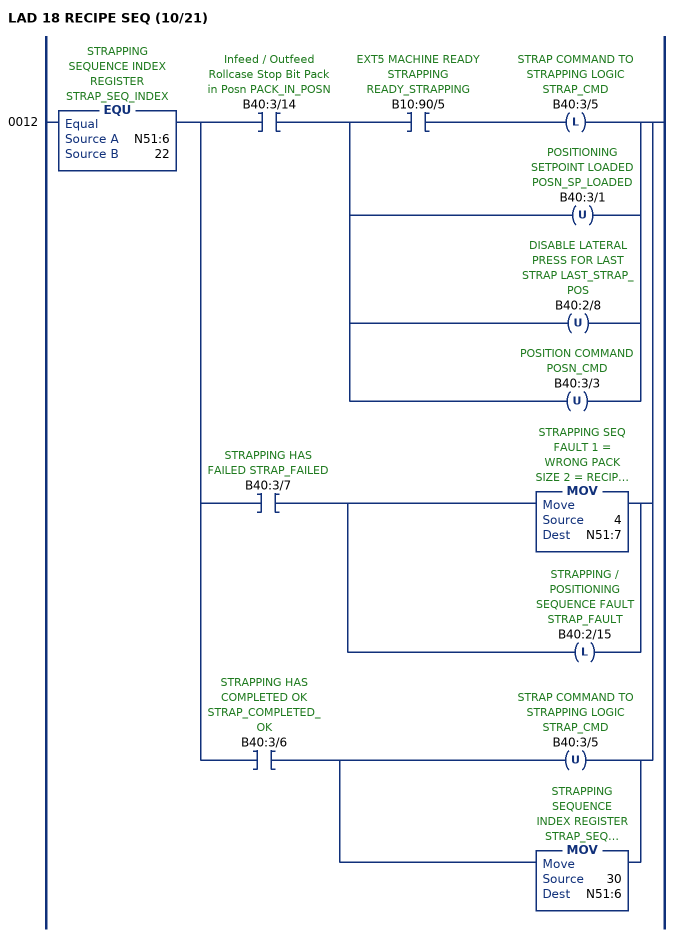
% Rung: 12 %
SOR EQU N51:6 22 BST XIC B40:3/14 BST XIC B10:90/5 OTL B40:3/5 NXB OTU B40:3/1 NXB OTU B40:2/8 NXB OTU B40:3/3 BND NXB XIC B40:3/7 BST MOV 4 N51:7 NXB OTL B40:2/15 BND NXB XIC B40:3/6 BST OTU B40:3/5 NXB MOV 30 N51:6 BND BND EOR
%   N51:6  STRAP_SEQ_INDEX  "STRAPPING SEQUENCE INDEX REGISTER" %
%   B40:3/14  PACK_IN_POSN  "Infeed / Outfeed Rollcase Stop Bit Pack in Posn" %
%   B10:90/5  READY_STRAPPING  "EXT5 MACHINE READY STRAPPING" %
%   B40:3/5  STRAP_CMD  "STRAP COMMAND TO STRAPPING LOGIC" %
%   B40:3/1  POSN_SP_LOADED  "POSITIONING SETPOINT LOADED" %
%   B40:2/8  LAST_STRAP_POS  "DISABLE LATERAL PRESS FOR LAST STRAP" %
%   B40:3/3  POSN_CMD  "POSITION COMMAND" %
%   B40:3/7  STRAP_FAILED  "STRAPPING HAS FAILED" %
%   N51:7  STRAP_SEQ_FLT  "STRAPPING SEQ FAULT 1 = WRONG PACK SIZE 2 = RECIPE FAULT 3 = POSNING FAULT 4 = STRAPPING FAULT" %
%   B40:2/15  STRAP_FAULT  "STRAPPING / POSITIONING SEQUENCE FAULT" %
%   B40:3/6  STRAP_COMPLETED_OK  "STRAPPING HAS COMPLETED OK" %

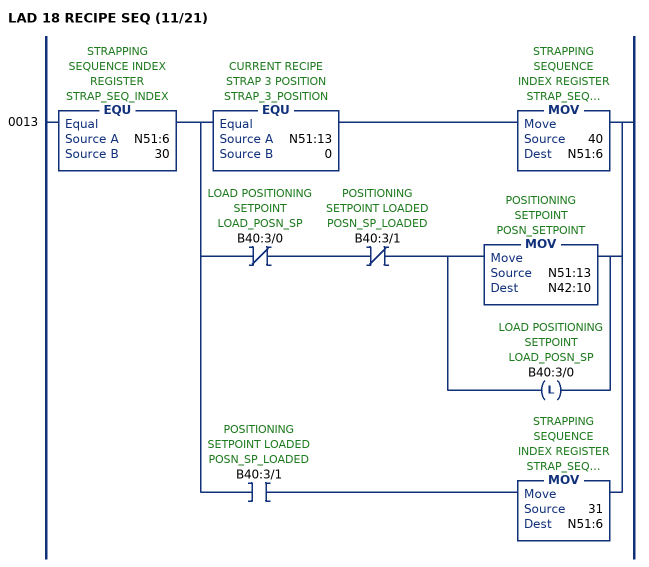
% Rung: 13 %
SOR EQU N51:6 30 BST EQU N51:13 0 MOV 40 N51:6 NXB XIO B40:3/0 XIO B40:3/1 BST MOV N51:13 N42:10 NXB OTL B40:3/0 BND NXB XIC B40:3/1 MOV 31 N51:6 BND EOR
%   N51:6  STRAP_SEQ_INDEX  "STRAPPING SEQUENCE INDEX REGISTER" %
%   N51:13  STRAP_3_POSITION  "CURRENT RECIPE STRAP 3 POSITION" %
%   B40:3/0  LOAD_POSN_SP  "LOAD POSITIONING SETPOINT" %
%   B40:3/1  POSN_SP_LOADED  "POSITIONING SETPOINT LOADED" %
%   N42:10  POSN_SETPOINT  "POSITIONING SETPOINT" %

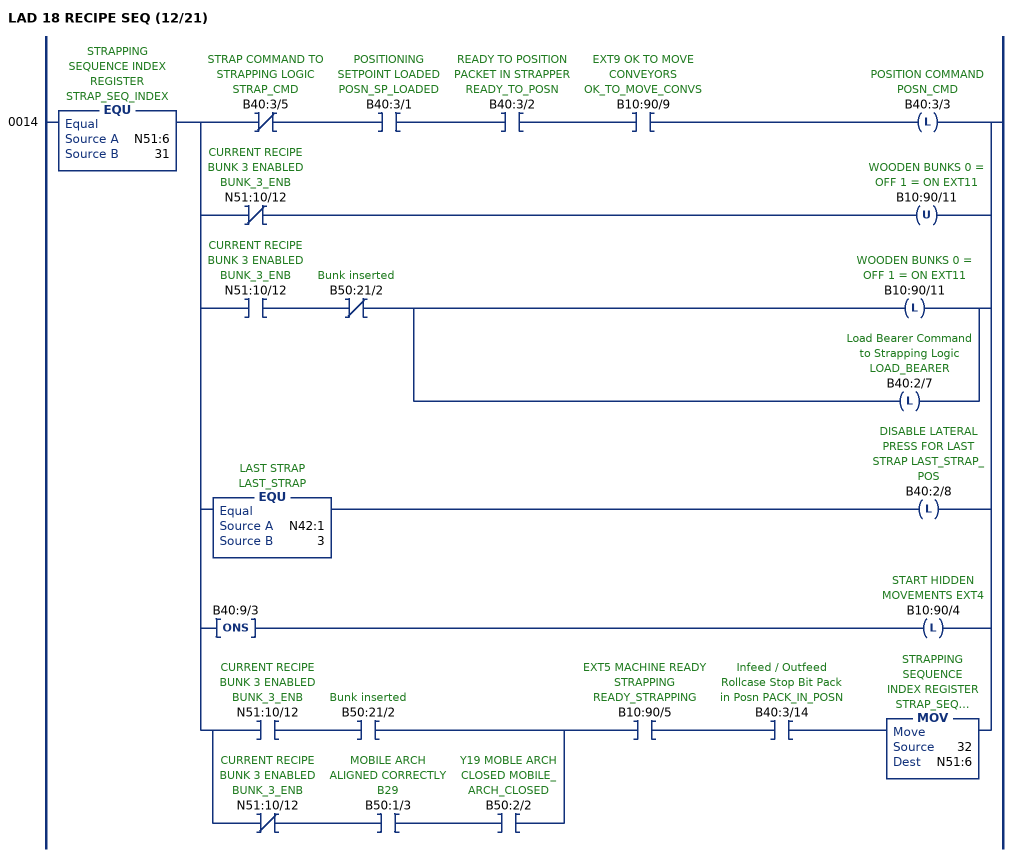
% Rung: 14 %
SOR EQU N51:6 31 BST XIO B40:3/5 XIC B40:3/1 XIC B40:3/2 XIC B10:90/9 OTL B40:3/3 NXB XIO N51:10/12 OTU B10:90/11 NXB XIC N51:10/12 XIO B50:21/2 BST OTL B10:90/11 NXB OTL B40:2/7 BND NXB EQU N42:1 3 OTL B40:2/8 NXB ONS B40:9/3 OTL B10:90/4 NXB BST XIC N51:10/12 XIC B50:21/2 NXB XIO N51:10/12 XIC B50:1/3 XIC B50:2/2 BND XIC B10:90/5 XIC B40:3/14 MOV 32 N51:6 BND EOR
%   N51:6  STRAP_SEQ_INDEX  "STRAPPING SEQUENCE INDEX REGISTER" %
%   B40:3/5  STRAP_CMD  "STRAP COMMAND TO STRAPPING LOGIC" %
%   B40:3/1  POSN_SP_LOADED  "POSITIONING SETPOINT LOADED" %
%   B40:3/2  READY_TO_POSN  "READY TO POSITION PACKET IN STRAPPER" %
%   B10:90/9  OK_TO_MOVE_CONVS  "EXT9 OK TO MOVE CONVEYORS" %
%   B40:3/3  POSN_CMD  "POSITION COMMAND" %
%   N51:10/12  BUNK_3_ENB  "CURRENT RECIPE BUNK 3 ENABLED" %
%   B10:90/11  EXT11  "WOODEN BUNKS 0 = OFF 1 = ON" %
%   B50:21/2  "Bunk inserted" %
%   B40:2/7  LOAD_BEARER  "Load Bearer Command to Strapping Logic" %
%   N42:1  LAST_STRAP  "LAST STRAP" %
%   B40:2/8  LAST_STRAP_POS  "DISABLE LATERAL PRESS FOR LAST STRAP" %
%   B10:90/4  EXT4  "START HIDDEN MOVEMENTS" %
%   B50:1/3  B29  "MOBILE ARCH ALIGNED CORRECTLY" %
%   B50:2/2  MOBILE_ARCH_CLOSED  "Y19 MOBLE ARCH CLOSED" %
%   B10:90/5  READY_STRAPPING  "EXT5 MACHINE READY STRAPPING" %
%   B40:3/14  PACK_IN_POSN  "Infeed / Outfeed Rollcase Stop Bit Pack in Posn" %

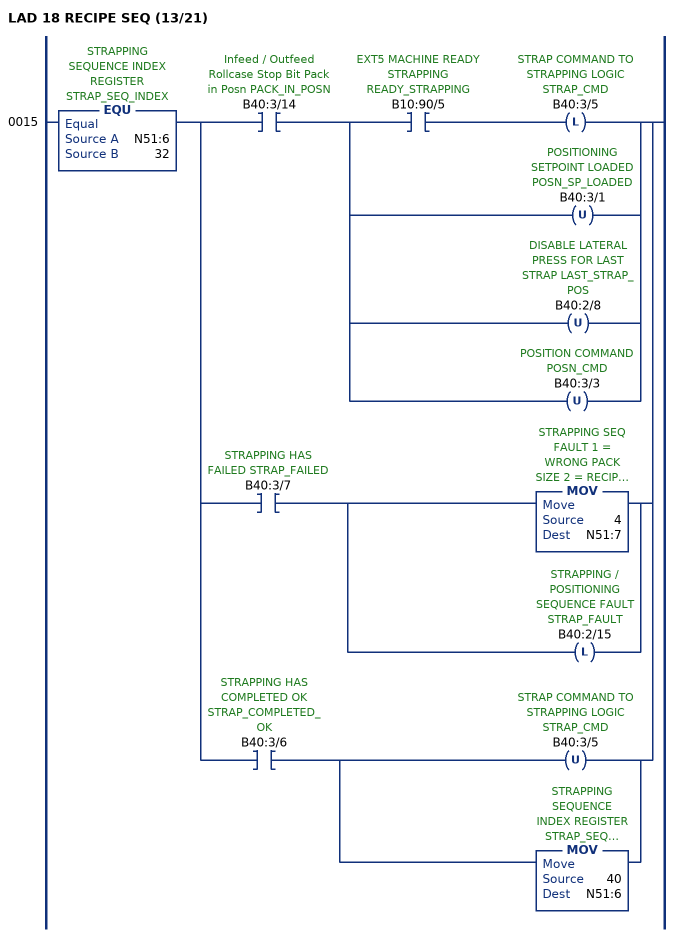
% Rung: 15 %
SOR EQU N51:6 32 BST XIC B40:3/14 BST XIC B10:90/5 OTL B40:3/5 NXB OTU B40:3/1 NXB OTU B40:2/8 NXB OTU B40:3/3 BND NXB XIC B40:3/7 BST MOV 4 N51:7 NXB OTL B40:2/15 BND NXB XIC B40:3/6 BST OTU B40:3/5 NXB MOV 40 N51:6 BND BND EOR
%   N51:6  STRAP_SEQ_INDEX  "STRAPPING SEQUENCE INDEX REGISTER" %
%   B40:3/14  PACK_IN_POSN  "Infeed / Outfeed Rollcase Stop Bit Pack in Posn" %
%   B10:90/5  READY_STRAPPING  "EXT5 MACHINE READY STRAPPING" %
%   B40:3/5  STRAP_CMD  "STRAP COMMAND TO STRAPPING LOGIC" %
%   B40:3/1  POSN_SP_LOADED  "POSITIONING SETPOINT LOADED" %
%   B40:2/8  LAST_STRAP_POS  "DISABLE LATERAL PRESS FOR LAST STRAP" %
%   B40:3/3  POSN_CMD  "POSITION COMMAND" %
%   B40:3/7  STRAP_FAILED  "STRAPPING HAS FAILED" %
%   N51:7  STRAP_SEQ_FLT  "STRAPPING SEQ FAULT 1 = WRONG PACK SIZE 2 = RECIPE FAULT 3 = POSNING FAULT 4 = STRAPPING FAULT" %
%   B40:2/15  STRAP_FAULT  "STRAPPING / POSITIONING SEQUENCE FAULT" %
%   B40:3/6  STRAP_COMPLETED_OK  "STRAPPING HAS COMPLETED OK" %

